{attribute 'signature_flag' := '1073741824'}
{attribute 'GUID' := '47DA0911-BC1D-4C26-A3DF-0D1E379DB03B'}
TYPE APICallMethod :
(
	GET,
    POST,
    PUT,
    DELETE,
    HEAD,
    OPTIONS,
    PATCH,
    MERGE,
    COPY
);
END_TYPE

(* stored: Version 1.1.0.1, ProductVersion 3.1.4022.12
   EnumerationTextList APICallMethod: Id {af99f943-4c71-4086-9aea-25ad92597d93} *)
